TYPE ST_SpecialTypes :
STRUCT
	NegativeIndexArray		: ARRAY[-100..100] OF LREAL := [1.11, 99(0.0), 5.55, 99(0.0), 9.99];
	MultiDimensionalArray	: ARRAY[1..3, 1..2] OF BYTE := [1, 2, 3, 4, 5, 6];
	ArrayOfArrays			: ARRAY[1..3] OF ARRAY[1..2] OF SINT := [[-1, -2], [-3, -4], [-5, -6]];
	
	PackMode1		: ST_StandardTypes_PackMode1;
	PackMode1_2		: ST_ComplexTypes_PackMode1;
	PackMode8		: ST_StandardTypes_PackMode8;
	PackMode8_2		: ST_ComplexTypes_PackMode8;
	
	EmptyBlock		: FB_EmptyBlock;
	EmptyStruct		: ST_EmptyStruct;
	EmptyArray 		: ARRAY[0..-1] OF BOOL; //How is this even possible..?
	
	Bits			: ST_Bits;
	
    {attribute 'TcEncoding':='UTF-8'}
	STRING_UTF8		: STRING := 'A test string ääöö!!@@';
END_STRUCT
END_TYPE

(* stored: Version 1.1.0.1, ProductVersion 3.1.4024.12
   DUT ST_SpecialTypes: Id {4e67e8d6-5a1e-4f09-805b-d0056fcc6955} *)
